// TIA Portal V18 export
TYPE "UDT_AHUsAI"
// stored: IsFailsafeCompliant false
   STRUCT
      rIAQ : Array[1..3] of Real;   // Рівень концентрації СО2 в торговій залі, ppm
      rBuildingdP : Array[1..3] of Real;   // Перепад тиску між будівлею і вулицею, Pa
      rRoomAirTemp_PLC_AI : Array[1..3] of Real;   // Температура повітря в торговій залі з вх PLC, C
      rSupplyAirTemp : Array[1..3] of Real;   // Температура повітря що подається з AHU в торгову залу, C
      rReturnAirTemp : Array[1..3] of Real;   // Температура повітря що подається з торгової зали в AHU, C
      rFrostProtWaterTemp : Array[1..3] of Real;   // Температура зворотнього теплоносія, C
      rFrostProtAirTemp : Array[1..3] of Real;   // Температура повытря пысля ТО, C x.50
      rRoomAirRelHumi : Array[1..3] of Real;
      rReserve : Array[1..3] of Real;   // Вулична температура x.99, C
      rSAFilterdP : Array[1..3] of Real;   // Перепад тиску на приточному filter x.53
      rSAFFlow : Array[1..3] of Real;   // Витрата повытря на припливному вентиляторы
      rRoomAirTemp_Actual : Array[1..3] of Real;   // Температура повітря в торговій залі Вираховане, C
      rRoomAirTemp_LoraAvg : Array[1..3] of Real;   // Температура повітря в торговій залі Вираховане, C
      rRoomAirTemp_MSensor : Array[1..3] of Real;   // Температура повітря в торговій залі Вираховане, C
      rReserve_1 : Array[1..3] of Real;
      rReserve_2 : Array[1..3] of Real;
      rReserve_3 : Array[1..3] of Real;
      rReserve_4 : Array[1..3] of Real;
      rReserve_5 : Array[1..3] of Real;
      rReserve_6 : Array[1..3] of Real;
      rReserve_7 : Array[1..3] of Real;
      rReserve_8 : Array[1..3] of Real;
      rReserve_9 : Array[1..3] of Real;
      cRoomTempSelect : Array[1..3] of Byte;   // 0=PLC_IO, 1=LoraAvg, 2=MSensor,3 =Auto
   END_STRUCT;
   // cRoomTempSelect[1] := 1;
   // cRoomTempSelect[2] := 0;
END_TYPE
